// TIA Portal V21 export
TYPE "LBC_typeAnalogScaleInterface"
TITLE = LBC_typeAnalogScaleInterface
// Module interface for external systems
   STRUCT
      commands : "LBC_typeInterfaceCommands";
      monitoring { ExternalWritable := 'False'} : "LBC_typeAnalogScaleValues";
      configuration : "LBC_typeAnalogScaleConfiguration";
   END_STRUCT;
END_TYPE
